{attribute 'linkalways'} 
{attribute 'no_explicit_call' := 'This FB is a CLASS and must be accessed using methods or properties'}
{attribute 'enable_dynamic_creation'}
FUNCTION_BLOCK _DWORD EXTENDS NumericDatatypeBase
VAR
	localData : DWORD;
	activeData : REFERENCE TO DWORD REF= localData;
END_VAR

PROPERTY PUBLIC Address : PVOID
GET
Address := ADR(activeData);
END_GET
END_PROPERTY

METHOD PUBLIC ClearReference
VAR_INPUT
END_VAR
activeData REF= localData;
END_METHOD

METHOD PUBLIC Clone : I_Datatype
VAR
    pClone : POINTER TO _DWORD;
END_VAR
pClone := __NEW(_DWORD(InitialValue := Value));
Clone := pClone^;
END_METHOD

METHOD FB_init : BOOL
VAR_INPUT
	bInitRetains : BOOL; // if TRUE, the retain variables are initialized (warm start / cold start)
	bInCopyCode : BOOL;  // if TRUE, the instance afterwards gets moved WORDo the copy code (online change)
	InitialValue : DWORD;
END_VAR
localData := InitialValue;
END_METHOD

PROPERTY PUBLIC IsFloat : BOOL
GET
IsFloat := FALSE;
END_GET
END_PROPERTY

PROPERTY PUBLIC IsSigned : BOOL
GET
IsSigned := FALSE;
END_GET
END_PROPERTY

PROPERTY PUBLIC LowerBound : DWORD
GET
LowerBound := DatatypeLimits.DWORD_LOWER_LIMIT;
END_GET
END_PROPERTY

METHOD PUBLIC MakeReferenceTo
VAR_INPUT
	ReferenceTarget : REFERENCE TO DWORD;
END_VAR
activeData REF= ReferenceTarget;
END_METHOD

METHOD PROTECTED SerializeLowerbound
VAR_INPUT
	Serializer : I_Serializer;
END_VAR
Serializer.AddDword(Lowerbound);
END_METHOD

METHOD PROTECTED SerializeUpperbound
VAR_INPUT
	Serializer : I_Serializer;
END_VAR
Serializer.AddDword(Upperbound);
END_METHOD

METHOD PUBLIC SerializeWith
VAR_INPUT
	Serializer : I_Serializer;
END_VAR
Serializer.AddDword(activeData);
END_METHOD

PROPERTY PUBLIC Size : UDINT
GET
Size := SIZEOF(activeData);
END_GET
END_PROPERTY

METHOD TryDeserializeFrom : BOOL
VAR_INPUT
	Deserializer : I_Deserializer;
	Feedback : I_DeserializerFeedback;
END_VAR
TryDeserializeFrom := Deserializer.TryGetDword(activeData, Feedback);
END_METHOD

METHOD TryMakeReferenceTo : BOOL
VAR_INPUT
	Target : I_Datatype;
END_VAR
VAR
	pTargetData : POINTER TO DWORD;
END_VAR
IF NOT (Target.TypeName = TypeName) THEN
	RETURN;
END_IF

pTargetData := Target.Address;
activeData REF= pTargetData^;
TryMakeReferenceTo := TRUE;
END_METHOD

PROPERTY PUBLIC TypeName : T_MAXSTRING
GET
TypeName := 'DWORD';
END_GET
END_PROPERTY

PROPERTY PUBLIC UpperBound : DWORD
GET
UpperBound := DatatypeLimits.DWORD_UPPER_LIMIT;
END_GET
END_PROPERTY

PROPERTY PUBLIC Value : DWORD
GET
Value := activeData;
END_GET
SET
activeData := Value;
END_SET
END_PROPERTY

END_FUNCTION_BLOCK

(* stored: Version 1.1.0.1, ProductVersion 3.1.4024.12
   POU _DWORD: Id {4c1cd110-10cf-0706-0267-224606ae6666}, SpecialFunc None
   Folder Constructor: Id {af0c863d-92bd-0c18-0dd4-64cc77b4094f}
   Folder Protected: Id {c3940d09-8489-0c0a-244d-316a1a31b5c9}
   Property Address: Id {9955f340-f87c-05a3-20a3-9824b3299552}
   Get Get: Id {a232f4f9-85cc-099b-2aa1-ea6f3b85eb4c}
   Method ClearReference: Id {964586d4-94ee-0de3-3238-dd792aac506c}
   Method Clone: Id {d6d02a4b-03e9-0ca2-0d51-7f2a9765df71}
   Method FB_init: Id {50a7d101-78a6-0e89-2f1d-c714c0dfe9cf}
   Property IsFloat: Id {ef056593-2728-0a16-21f3-fcca2e31797a}
   Get Get: Id {623d3531-b500-0648-04c7-82eda81aaffe}
   Property IsSigned: Id {133c0f05-fd33-0aaf-1027-972052ce4659}
   Get Get: Id {c61474ec-13e7-07b8-0cb1-b7ad40382560}
   Property LowerBound: Id {0cc28ba6-6da2-08ae-2b4c-4fdd65f9ea1a}
   Get Get: Id {5544e0a5-7db7-0166-317a-b8c312b3fae7}
   Method MakeReferenceTo: Id {cddf2b40-abe8-0141-3a14-a0695f4c6b1c}
   Method SerializeLowerbound: Id {608aece2-9605-00b2-209d-8ec3580a1f1f}
   Method SerializeUpperbound: Id {37aa899d-501e-01d9-1d08-71d728c3a8d2}
   Method SerializeWith: Id {eb21cfdd-f895-0d4a-278c-25149b1f23a5}
   Property Size: Id {cb4e3165-7d10-06fc-2e94-5a3e0597f98b}
   Get Get: Id {9a624e2f-adae-0cc4-1b24-57c8307dbc4c}
   Method TryDeserializeFrom: Id {c1d63ad7-1231-0bdb-2694-0779ce112455}
   Method TryMakeReferenceTo: Id {01274e6c-9478-014b-10d8-8a050477d8ff}
   Property TypeName: Id {2d24b760-237b-08cb-1293-75cc3e2d65cc}
   Get Get: Id {39e29c35-93a9-0ffa-05ce-2a16e047a297}
   Property UpperBound: Id {414981f6-6ae5-0924-2010-f24015c2a17b}
   Get Get: Id {c3b206e2-ad02-0685-02ba-8095be503eef}
   Property Value: Id {bfcf5460-41d4-07cb-2a79-70b2be60af8f}
   Get Get: Id {7b37ae66-753a-095a-2266-5ed4c94ddb63}
   Set Set: Id {42349c48-093b-0e01-056c-ae500413f5f0} *)
